Universal Robots PolyScope program: _adminCG-InvAtoPHome.urp

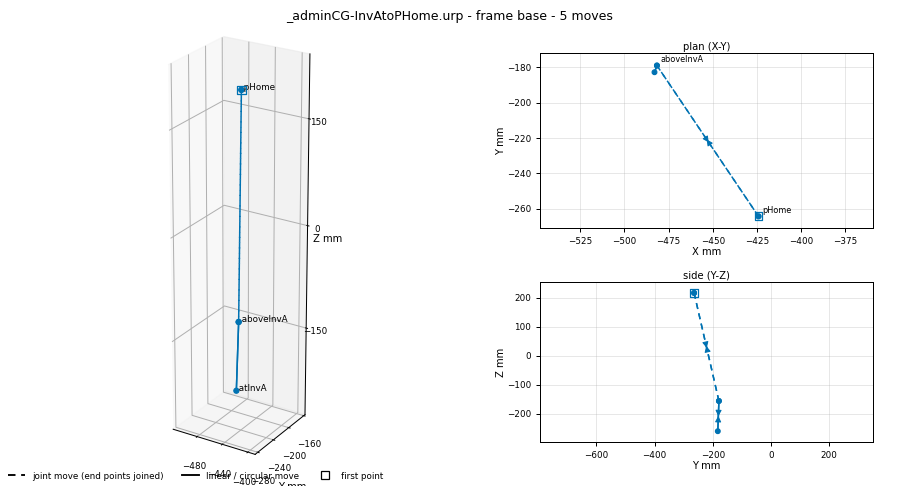
[picture p0: tool path of _adminCG-InvAtoPHome.urp in frame base, 5 of 5 moves have a stored position in this frame; points joined in program order, loops and branches not executed]
Program _adminCG-InvAtoPHome (installation=admin directory=/programs/THU_530PM createdIn=3.15.8.106339 lastSavedIn=3.15.8.106339 robotSerialNumber=2015350925)
Calibrated DH parameters: a=[0, -0.425, -0.39225, 0, 0, 0]; d=[0.089159, 0, 0, 0.10915, 0.09465, 0.0823]; alpha=[1.570796, 0, 0, 1.570796, -1.570796, 0]; deltaTheta=[0, 0, 0, 0, 0, 0]
Robot Program (runOnlyOnce=true)
  Set DigitalOutput pin=digital_out[0]; digitalValue=0
  Call _adminLinearIndex1
  MoveJ speed 60 deg/s, acceleration 80 deg/s^2 (useActiveTCP=true)
    Waypoint pHome: TCP in base x=-424.178 y=-264.255 z=215.89 mm, rx=-1.1973 ry=-2.8916 rz=-0.0084 rad; joints [224.995, -90.004, -90.004, -90.016, 89.253, -0.021] deg; flange x=-422.252 y=-266.309 z=431.771 mm, rx=-1.1973 ry=-2.8916 rz=-0.0084 rad
    Waypoint aboveInvA: TCP in base x=-481.65 y=-178.932 z=-155.682 mm, rx=-1.1941 ry=-2.8953 rz=-0.0079 rad; joints [213.016, -116.521, -119.972, -33.429, 89.376, -12.161] deg; flange x=-480.123 y=-180.743 z=60.205 mm, rx=-1.1941 ry=-2.8953 rz=-0.0079 rad
  MoveL speed 250 mm/s, acceleration 1200 mm/s^2 (useActiveTCP=true) feature=Base
    Waypoint atInvA: TCP in base x=-483.023 y=-182.727 z=-259.58 mm, rx=-1.1934 ry=-2.896 rz=-0.0068 rad; joints [213.266, -131.209, -119.597, -19.098, 89.419, -11.943] deg; flange x=-481.522 y=-184.358 z=-43.692 mm, rx=-1.1934 ry=-2.896 rz=-0.0068 rad
    Set DigitalOutput pin=digital_out[0]; digitalValue=1
    Wait Sleep waitTime=1
    Waypoint aboveInvA: TCP in base x=-481.65 y=-178.932 z=-155.682 mm, rx=-1.1941 ry=-2.8953 rz=-0.0079 rad; joints [213.016, -116.521, -119.972, -33.429, 89.376, -12.161] deg; flange x=-480.123 y=-180.743 z=60.205 mm, rx=-1.1941 ry=-2.8953 rz=-0.0079 rad
  MoveJ speed 60 deg/s, acceleration 80 deg/s^2 (useActiveTCP=true)
    Waypoint pHome: TCP in base x=-424.178 y=-264.255 z=215.89 mm, rx=-1.1973 ry=-2.8916 rz=-0.0084 rad; joints [224.995, -90.004, -90.004, -90.016, 89.253, -0.021] deg; flange x=-422.252 y=-266.309 z=431.771 mm, rx=-1.1973 ry=-2.8916 rz=-0.0084 rad
SubProgram -> _adminLinearIndex1
SubProgram _adminLinearIndex1 (keepSynchronizedWithDisk=false) programFile=/programs/me345_admin/_adminLinearIndex1.urp
  Folder Move_linear_slide_Index1
    var_1 := False
    Loop While (checkContinuously=false) expression=var_1≟ False
      var_1 := socket_open("10.241.34.48",4001)
    var_3 := 1
    Send := "s r0x24 21"
    Script: socket_send_string(Send)
    Script: socket_send_byte(13)
    Send_Reply := socket_read_string()
    Send := "s r0xca 0"
    Script: socket_send_string(Send)
    Script: socket_send_byte(13)
    Send_Reply := socket_read_string()
    Send := "t 1"
    Script: socket_send_string(Send)
    Script: socket_send_byte(13)
    Send_Reply := socket_read_string()
    Loop While (checkContinuously=false) expression=var_3≠0
      Send := "g r0xA0"
      Script: socket_send_string(Send)
      Script: socket_send_byte(13)
      var_3 := socket_get_var("v")
      Wait Sleep waitTime=0.1
    Script: socket_close()
    Script: sync()
